Staubli VAL3: makeTraj.pgx

program makeTraj(num x_nJointStart, string x_sTrajLoad)
  local num i
  local bool l_bToStop[2]
  local num l_nSize
  local tool l_tTool
  local num l_nSpeed[2]
  local mdesc l_mDesc[2]
  local num l_nDistance[2]
  local num l_nMoveType[2]
  local point l_pAction
  local bool l_bUnreached
  local num l_nStop
  local point l_pCheck[3]
  local point l_pHere
  local frame l_fPlane
  local num l_nTime
  local string l_sType
  local string l_sMessage
  local bool l_bConnection
  local num l_nMoveId
  local TrajectoryItem l_tTraj
  local joint l_jJoint
  local ActionItem l_aAction
  local num j
  local bool l_bGoToCloseP
  local point l_pHereJ
  local joint l_jResult
  local bool l_bOk
  local num i_from
  local num i_to
  local joint l_jHere
  local joint l_jRunJoint[2]
begin
  //
  // inizialize the system
  //
  // use the flange
  l_tTool=flange
  // the maximum size
  call getSizeItem(true,l_nSize)
  //
  // first go near by straight line of the two previous points
  //
  if pt:tTraj[sTrajCycle].nZoneType!=0 and x_nJointStart==0
    // use of the ZONE TYPE
    switch pt:tTraj[sTrajCycle].nZoneMove
      case 0
        l_sType="POINT"
      break
      case 1
        l_sType="APPRO"
      break
      case 2
        l_sType="Z VALUE"
      break
      case 3
        l_sType="@Point"
      break
      case 4
        l_sType="@JPoint"
      break
    endSwitch
    cycleStatus:sToShow="Move using: "+l_sType+toString("",x_nJointStart)+"# of the home: "+x_sTrajLoad
    logMsg("HOMING: "+l_sMessage)
    call getPointData(l_nSpeed,l_mDesc,l_nDistance,l_bToStop,l_nMoveType,l_nStop,0,true)
    call moveTo(l_tTool,l_mDesc,l_nMoveType,l_bUnreached,0,l_nMoveId,true)
    waitEndMove()
    // set the start point
    x_nJointStart=1
  elseIf saveData:bUseHomeScanner
    // look FORWARD
    if x_nJointStart<l_nSize-1
      // get all the JOINT
      call getJointData(l_jRunJoint[0],l_tTool,true,x_nJointStart+1)
      call getJointData(l_jRunJoint[1],l_tTool,true,x_nJointStart)
      // look if there is
      if setFrame(jointToPoint(l_tTool,world,l_jRunJoint[0]),jointToPoint(l_tTool,world,l_jRunJoint[1]),pNull,fFrame)==0
        pCheck=here(l_tTool,fFrame)
        if pCheck.trsf.x>=0
          //
          // go to nearest point
          //
          call getPoint(l_pCheck[0],true,x_nJointStart+1)
          call getPoint(l_pCheck[1],true,x_nJointStart)
          x_nJointStart=x_nJointStart+1
          l_bGoToCloseP=true
        endIf
      endIf
    endIf
    // LOOK BACKWARD
    if !l_bGoToCloseP and x_nJointStart>0
      // get all the JOINT
      call getJointData(l_jRunJoint[0],l_tTool,true,x_nJointStart)
      call getJointData(l_jRunJoint[1],l_tTool,true,x_nJointStart-1)
      // look if there is
      if setFrame(jointToPoint(l_tTool,world,l_jRunJoint[0]),jointToPoint(l_tTool,world,l_jRunJoint[1]),pNull,fFrame)==0
        pCheck=here(l_tTool,fFrame)
        if pCheck.trsf.x>=0
          //
          // go to nearest point
          //
          call getPoint(l_pCheck[0],true,x_nJointStart)
          call getPoint(l_pCheck[1],true,x_nJointStart-1)
          l_bGoToCloseP=true
        endIf
      endIf
    endIf
    // go to an approach POINT
    if l_bGoToCloseP
      // init
      l_pCheck[2]=here(l_tTool,world)
      l_pHere=here(l_tTool,world)
      l_pHereJ=here(flange,world)
      l_nDistance=10000
      // check the nearest point
      l_nMoveType=pt:tTraj[sTrajCycle].tData[x_nJointStart].tSuper.moveType
      for i=0 to 1 step 0.1
        if l_nMoveType==0
          call interpolateJ(l_jRunJoint[1],l_jRunJoint[0],i,l_jResult,l_bOk)
          l_pCheck[2]=jointToPoint(flange,world,l_jResult)
          if l_nDistance>=distance(l_pCheck[2],l_pHereJ)
            l_nDistance=distance(l_pCheck[2],l_pHereJ)
            //save the value
            l_nStop=i
          endIf
        else
          l_pCheck[2].trsf=interpolateL(l_pCheck[1].trsf,l_pCheck[0].trsf,i)
          l_bOk=true
          if l_nDistance>=distance(l_pCheck[2],l_pHere)
            l_nDistance=distance(l_pCheck[2],l_pHere)
            //save the value
            l_nStop=i
          endIf
        endIf
      endFor
      // closer search
      i_from=(max(l_nStop-0.05,0))
      i_to=(min(l_nStop+0.05,1))
      for i=i_from to i_to step 0.01
        if l_nMoveType==0
          call interpolateJ(l_jRunJoint[1],l_jRunJoint[0],i,l_jResult,l_bOk)
          l_pCheck[2]=jointToPoint(flange,world,l_jResult)
          if l_nDistance>=distance(l_pCheck[2],l_pHereJ)
            l_nDistance=distance(l_pCheck[2],l_pHereJ)
            //save the value
            l_nStop=i
          endIf
        else
          l_pCheck[2].trsf=interpolateL(l_pCheck[1].trsf,l_pCheck[0].trsf,i)
          l_bOk=true
          if l_nDistance>=distance(l_pCheck[2],l_pHere)
            l_nDistance=distance(l_pCheck[2],l_pHere)
            //save the value
            l_nStop=i
          endIf
        endIf
      endFor
      // set the best one
      call getPointData(l_nSpeed,l_mDesc,l_nDistance,l_bToStop,l_nMoveType,l_nStop,x_nJointStart,true)
      l_jHere=herej()
      if l_nMoveType==0
        call interpolateJ(l_jRunJoint[1],l_jRunJoint[0],l_nStop,l_jResult,l_bOk)
        l_pCheck[2]=jointToPoint(flange,world,l_jResult)
        // put the wrist on free
        l_pCheck[2].config.wrist=wfree
        if pointToJoint(l_tTool,herej(),l_pCheck[2],l_jHere)
          movej(l_pCheck[2],flange,l_mDesc)
        endIf
      else
        l_pCheck[2].trsf=interpolateL(l_pCheck[1].trsf,l_pCheck[0].trsf,l_nStop)
        // put the wrist on free
        l_pCheck[2].config.wrist=wfree
        if pointToJoint(l_tTool,herej(),l_pCheck[2],l_jHere)
          movej(l_pCheck[2],l_tTool,l_mDesc)
        endIf
      endIf
      // show the message
      cycleStatus:sToShow="Move to point: "+toString("",x_nJointStart+1)+" of: "+x_sTrajLoad +" % "+toString(".3",l_nStop)
      logMsg("HOMING: "+cycleStatus:sToShow)
      waitEndMove()
    endIf
  endIf
  //
  // for all of my traj cyclePoints move the robot
  //
  resize(tTraj.tSuper,1,size(pt:tTraj[sTrajCycle].tData))
  for i=x_nJointStart to (l_nSize-1)
    tTraj.tSuper[i]=pt:tTraj[sTrajCycle].tData[i].tSuper
  endFor
  tTraj.sID="HOME "+pt:tTraj[sTrajCycle].sID
  call cycleStatus:addTraj(tTraj)
  // show the message
  cycleStatus:sToShow="Moving from point: "+toString("",x_nJointStart+1)+" of : "+x_sTrajLoad
  logMsg("HOMING: "+cycleStatus:sToShow)
  for i=x_nJointStart to (l_nSize-1)
    //
    // get the point info
    //
    l_tTraj=pt:tTraj[sTrajCycle].tData[i].tSuper
    //
    // get the distance in percentage
    //
    call getDistance(l_tTool,l_nDistance,true,i)
    //
    // give to the traj library the percentage distance
    //
    if l_tTraj.toStop
      l_tTraj.nom_speed.blend=off
    endIf
    //
    // put the move in the stack
    //
    l_jJoint=pt:tTraj[sTrajCycle].tData[i].jJoint
    call moveTo(l_tTool,l_tTraj.nom_speed,l_tTraj.moveType,l_bUnreached,i,l_nMoveId,true)
    // set the data
    l_aAction.nDistance=l_nDistance
    l_aAction.nPointId=i
    l_aAction.nMoveId=l_nMoveId
    l_aAction.sIdTraj="HOME "+pt:tTraj[sTrajCycle].sID
    call cycleStatus:putInstr_Traj(l_aAction,l_tTraj,pt:tTraj[sTrajCycle].nIndexTool,l_nSize)
    // there is a waitEndMove
    if l_tTraj.toStop
      waitEndMove()
      delay(l_tTraj.nStop)
      // wait all the action has been done
      wait(cycleStatus:bActionRunning==false)
    endIf
  endFor
end
